INTERFACE I_ListString EXTENDS I_ListBase

METHOD PUBLIC M_Remove : BOOL
VAR_INPUT
	Object: 	STRING(255);
END_VAR
END_METHOD

METHOD PUBLIC M_Index : STRING(255)
VAR_INPUT
	Index: 	DINT;
END_VAR
END_METHOD

METHOD PUBLIC M_Find : DINT
VAR_INPUT
	Object: 	STRING(255);
END_VAR
END_METHOD

METHOD PUBLIC M_Add : BOOL
VAR_INPUT
	Object: 	STRING(255);
END_VAR
END_METHOD

END_INTERFACE

(* stored: Version 1.1.0.1
   Itf I_ListString: Id {95dd71be-3dad-41c6-ba89-70dc44fa9415}
   Method M_Remove: Id {651ced80-bc93-40fe-9ff8-dfe0a20c890e}
   Method M_Index: Id {6e7d021b-fda4-4baf-9fa0-4eab4b7b6b25}
   Method M_Find: Id {a10273cc-82fe-44c2-b72a-533847e41f69}
   Method M_Add: Id {b1ced62e-04c6-447f-96b8-b1c7d3454f6a} *)
